// TIA Portal V19 export
DATA_BLOCK "TRK_Info"   // DB186
// stored: Access Published, MemoryReserve 100
   VAR
      HMI_Info : "BTrk_item";
   END_VAR
BEGIN
END_DATA_BLOCK
